% RSLogix 500 project P3 - Inventory Management.RSS, saved by version 8.30.00.16 %
PROJECT "PROJECT3"    % processor: Bul.1763 MicroLogix 1100 Series B %

PROGRAM FILES
  LAD 2 "MAIN"  6 rungs
  LAD 3 "QUANTITY"  6 rungs
  LAD 4 "RESET"  3 rungs

DATA FILES
  O0 OUTPUT  4 elements
  I1 INPUT  6 elements
  S2 STATUS  66 elements
  B3 BINARY  1 elements
  T4 TIMER  1 elements
  C5 COUNTER  1 elements
  R6 CONTROL  1 elements
  N7 INTEGER  10 elements
  F8 FLOAT  1 elements
  ST9 STRING  10 elements

LADDER 2 "MAIN"
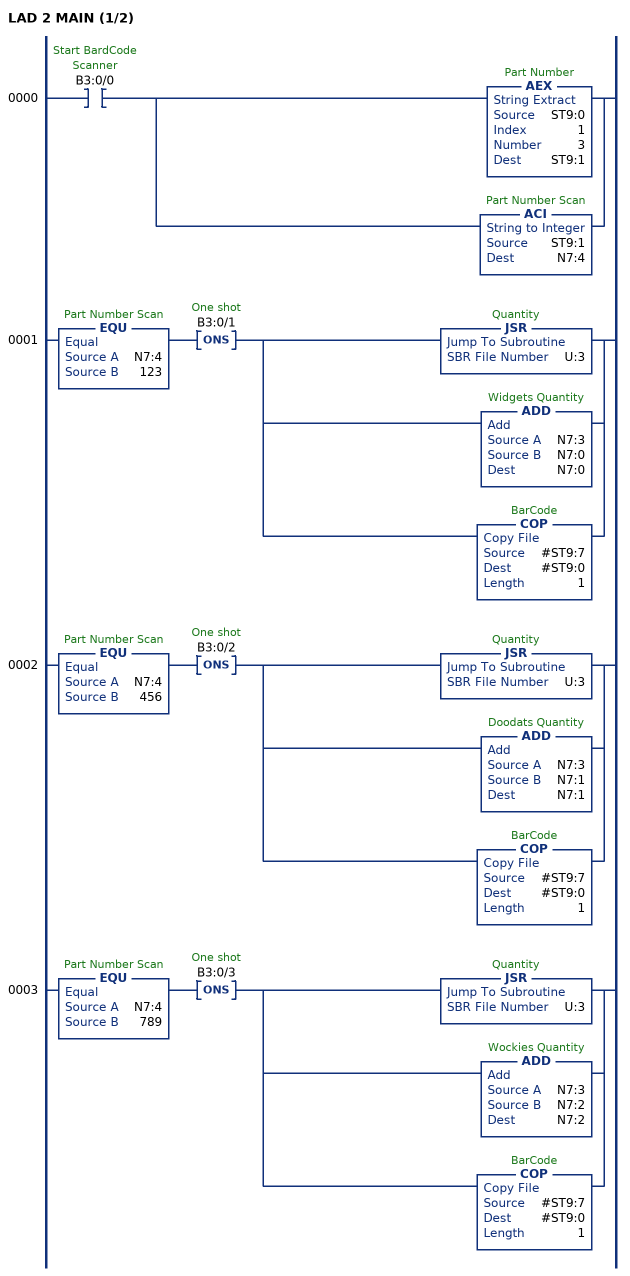
% Rung: 0 %
SOR XIC B3:0/0 BST AEX ST9:0 1 3 ST9:1 NXB ACI ST9:1 N7:4 BND EOR
%   B3:0/0  "Start BardCode Scanner" %
%   ST9:0  "BarCode" %
%   ST9:1  "Part Number" %
%   N7:4  "Part Number Scan" %
% Rung: 1 %
SOR EQU N7:4 123 ONS B3:0/1 BST JSR U:3 NXB BST ADD N7:3 N7:0 N7:0 NXB COP #ST9:7 #ST9:0 1 BND BND EOR
%   N7:4  "Part Number Scan" %
%   B3:0/1  "One shot" %
%   U:3  "Quantity" %
%   N7:3  "Quantity Adder" %
%   N7:0  "Widgets Quantity" %
%   ST9:0  "BarCode" %
% Rung: 2 %
SOR EQU N7:4 456 ONS B3:0/2 BST JSR U:3 NXB BST ADD N7:3 N7:1 N7:1 NXB COP #ST9:7 #ST9:0 1 BND BND EOR
%   N7:4  "Part Number Scan" %
%   B3:0/2  "One shot" %
%   U:3  "Quantity" %
%   N7:3  "Quantity Adder" %
%   N7:1  "Doodats Quantity" %
%   ST9:0  "BarCode" %
% Rung: 3 %
SOR EQU N7:4 789 ONS B3:0/3 BST JSR U:3 NXB ADD N7:3 N7:2 N7:2 NXB COP #ST9:7 #ST9:0 1 BND EOR
%   N7:4  "Part Number Scan" %
%   B3:0/3  "One shot" %
%   U:3  "Quantity" %
%   N7:3  "Quantity Adder" %
%   N7:2  "Wockies Quantity" %
%   ST9:0  "BarCode" %

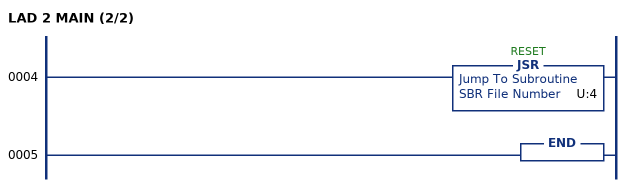
% Rung: 4 %
SOR JSR U:4 EOR
%   U:4  "RESET" %
% Rung: 5 %
SOR END EOR

LADDER 3 "QUANTITY"
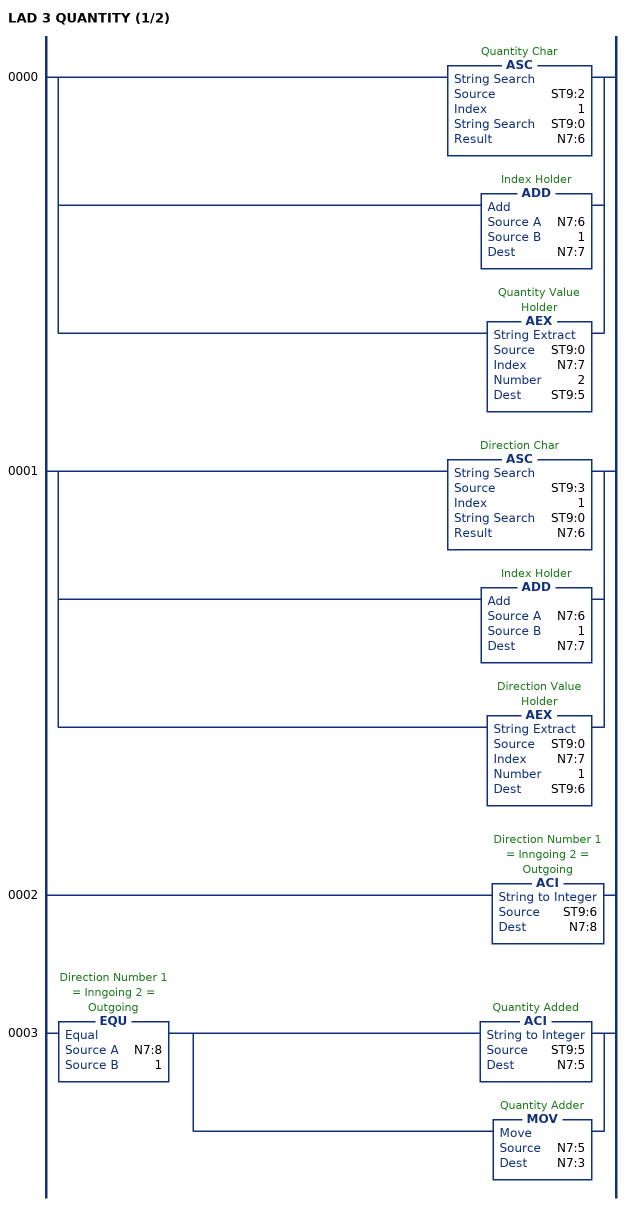
% Rung: 0 %
SOR BST ASC ST9:2 1 ST9:0 N7:6 NXB BST ADD N7:6 1 N7:7 NXB AEX ST9:0 N7:7 2 ST9:5 BND BND EOR
%   ST9:2  "Quantity Char" %
%   ST9:0  "BarCode" %
%   N7:6  "QQ number" %
%   N7:7  "Index Holder" %
%   ST9:5  "Quantity Value Holder" %
% Rung: 1 %
SOR BST ASC ST9:3 1 ST9:0 N7:6 NXB BST ADD N7:6 1 N7:7 NXB AEX ST9:0 N7:7 1 ST9:6 BND BND EOR
%   ST9:3  "Direction Char" %
%   ST9:0  "BarCode" %
%   N7:6  "QQ number" %
%   N7:7  "Index Holder" %
%   ST9:6  "Direction Value Holder" %
% Rung: 2 %
SOR ACI ST9:6 N7:8 EOR
%   ST9:6  "Direction Value Holder" %
%   N7:8  "Direction Number 1 = Inngoing 2 = Outgoing" %
% Rung: 3 %
SOR EQU N7:8 1 BST ACI ST9:5 N7:5 NXB MOV N7:5 N7:3 BND EOR
%   N7:8  "Direction Number 1 = Inngoing 2 = Outgoing" %
%   ST9:5  "Quantity Value Holder" %
%   N7:5  "Quantity Added" %
%   N7:3  "Quantity Adder" %

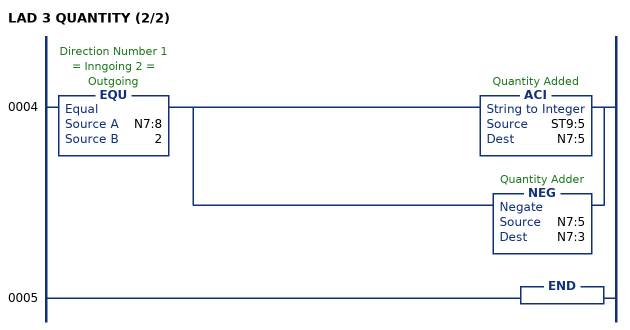
% Rung: 4 %
SOR EQU N7:8 2 BST ACI ST9:5 N7:5 NXB NEG N7:5 N7:3 BND EOR
%   N7:8  "Direction Number 1 = Inngoing 2 = Outgoing" %
%   ST9:5  "Quantity Value Holder" %
%   N7:5  "Quantity Added" %
%   N7:3  "Quantity Adder" %
% Rung: 5 %
SOR END EOR

LADDER 4 "RESET"
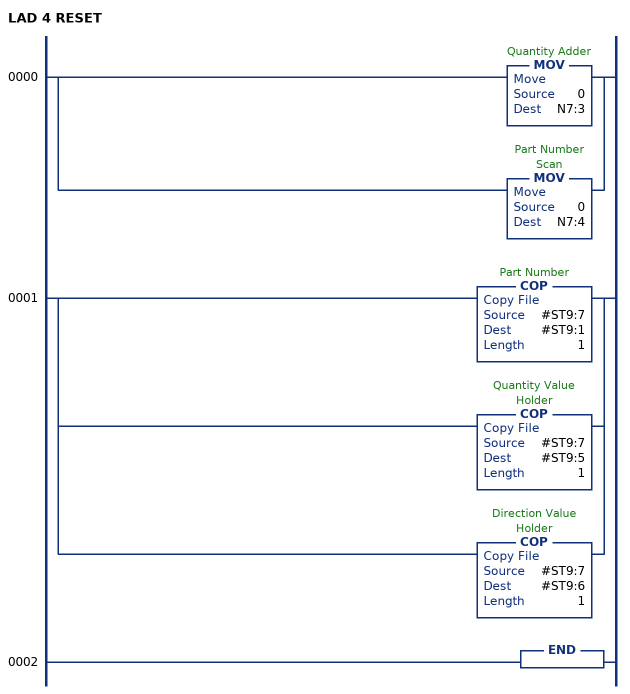
% Rung: 0 %
SOR BST MOV 0 N7:3 NXB MOV 0 N7:4 BND EOR
%   N7:3  "Quantity Adder" %
%   N7:4  "Part Number Scan" %
% Rung: 1 %
SOR BST COP #ST9:7 #ST9:1 1 NXB COP #ST9:7 #ST9:5 1 NXB COP #ST9:7 #ST9:6 1 BND EOR
%   ST9:1  "Part Number" %
%   ST9:5  "Quantity Value Holder" %
%   ST9:6  "Direction Value Holder" %
% Rung: 2 %
SOR END EOR

OTHER DOCUMENTED ADDRESSES
  B3:0/4  "one shot"
  B3:0/5  "Reset Trigger"
  Q0:0  "d"
  ST9:7.0  "Empty String"
  T4:0  "Quantity Timer Delay"

DATA TABLE (non-zero values as saved)
DATA B3
% B3:0 % 0X0008
DATA T4
% .PRE .ACC %
% T4:0 % 3 0
DATA ST9
% ST9:0 % "PPP-QQ:D"
% ST9:2 % "-"
% ST9:3 % ":"
